TYPE U_FanucCNCEventSourceInfo :
UNION
	{attribute 'displaymode':='hex'}
	Id : DWORD;
	Details : ST_FanucCNCEventSourceDetails;
END_UNION

END_TYPE

(* stored: Version 1.1.0.1, ProductVersion 3.1.4024.12
   DUT U_FanucCNCEventSourceInfo: Id {222bd233-f168-4d4b-8c8b-277714ef5572} *)
